(*
Copyrights	: Precision Systems Engineering
Author		: ADBO
Date		: 07/2022
Description	: This function block extends standard functionality of FB_FixtureCore with platform pusher and product holder.
*)
FUNCTION_BLOCK FB_Fixture EXTENDS FB_FixtureJig
VAR CONSTANT
	(* Fixture platform cylinder default setup *)
	sCOVER_PUSHER_NAME						: STRING	:= 'Cover Pusher';	(* Platform pusher name *)
	tCOVER_PUSHER_OPEN_TIMEOUT				: TIME 		:= T#5S;			(* Platform pusher opening timeout *)
	tCOVER_PUSHER_CLOSE_TIMEOUT				: TIME 		:= T#5S;			(* Platform pusher closing timeout *)
	tCOVER_PUSHER_MOVE_DELAY 				: TIME 		:= T#0MS;			(* Platform pusher delay after position change *)
	
	(* Fixture product holder default setup *)
	sCLAMP_NAME								: STRING 	:= 'Clamp Pusher';	(* Product holder name *)
	tCLAMP_OPEN_TIMEOUT						: TIME 		:= T#5S;			(* Product holder opening timeout *)
	tCLAMP_CLOSE_TIMEOUT					: TIME 		:= T#5S;			(* Product holder closing timeout *)
	tCLAMP_MOVE_DELAY 						: TIME 		:= T#300MS;//750MS	(* Product holder delay after position change *)
	
	(* Norm loading keywords *)
	sNORM_LOAD_COMMAND						: STRING := 'LDNORM:';			(* Load norm command send from PLC to UTU*)
	sNORM_GSAMPLE_MEASURE_COMMAND			: STRING := 'MeasGSample';		(* Measure Golden sample command send from PLC to UTU after loading new norm *)	
	sNORM_LOAD_SUCCESS 						: STRING := 'OK';				(* Response from UTU: norm loaded successfull *)
	sNORM_LOAD_FAIL							: STRING := 'Fail';				(* Response from UTU: norm load failed *)
	sNORM_GS_REQUEST						: STRING := 'GS:';				(* UTU requests golden sample *)
 	
	(* UTU STATUS *)
	sUTU_STATUS_OK							: STRING := 'OK';
	sUTU_STATUS_NOK							: STRING := 'NOK';
	sUTU_STATUS_bBusy						: STRING := 'bBusy';
	sUTU_STATUS_BCHECKSETUP					: STRING := 'bCheckSetup';
	
	(* Measurement keywords *)
	sMEASUREMENT_START_COMMAND				: STRING := 'bStart$R$N';		(* Start measurement command send from PLC to UTU*)
	
	sMEASUREMENT_BUSY						: STRING := 'bBusy';			(* Response from UTU: measurement started *)
	sMEASUREMENT_FINISHED					: STRING := (*'bReady'; //*)'bDone';			(* Response from UTU: measurement passed *)
	sMEASUREMENT_GOOD_PRODUCT				: STRING := 'bGood';			(* Response from UTU: good product *)
	sMEASUREMENT_REWORK						: STRING := 'bRework';			(* Perform remeasurement of same product *)
	sMEASUREMENT_REMEASURE					: STRING := 'bRemeasure';		(* Perform remeasurement of same product *)
	sMEASUREMENT_ERROR_THD					: STRING := 'bTHDReject';		(* Response from UTU: measurement failed with THD error*)
	sMEASUREMENT_ERROR_PHASE				: STRING := 'bPhaseReject';		(* Response from UTU: measurement failed with PHASE error*)
	sMEASUREMENT_ERROR_SSPL					: STRING := 'bSSPLReject';		(* Response from UTU: measurement failed with SSPL error*)
	sMEASUREMENT_ERROR_RUBBING				: STRING := 'bRubReject';		(* Response from UTU: measurement failed with RUBBING error*)
	sMEASUREMENT_ERROR_IMP					: STRING := 'bImpReject';		(* Response from UTU: measurement failed with INP error*)
	sMEASUREMENT_ERROR_HFA					: STRING := 'bHFAReject';		(* Response from UTU: measurement failed with HFA error*)
	sMEASUREMENT_ERROR_SPL					: STRING := 'bSPLReject';		(* Response from UTU: measurement failed with SPL error*)
	sMEASUREMENT_ERROR_CONNECTION			: STRING := 'bRejectConnect';	(* Response from UTU: measurement failed with connection problems *)
	sMEASUREMENT_ERROR_OTHER				: STRING := 'bReject';			(* Response from UTU: measurement failed *)
	sMEASUREMENT_FINISH_BATCH				: STRING := 'bFinishBatch';		(* Response from UTU: Batch END *)
	sMEASUREMENT_READY						: STRING := 'bReady';
END_VAR
VAR
	(* Auxilary command bits *)
	bCoverActive 							: BOOL;
	bCoverHome 								: BOOL;
	bClampHold 								: BOOL;
	bClampRelease 							: BOOL;
	bCoverActiveAndJigOpen					: BOOL;
	bCoverHomeAndJigClose					: BOOL;
	bLoadNorm								: BOOL;
//	bGSampleMeasure							: BOOL;
//	bGoldenSampelReadyToMeasure				: BOOL;		(* Robot gived Golden sample to Fixture *)
	
	(* Parameters *)
	sProductType							: STRING;
	sProductQuantity						: STRING;
	
	//new
	sConfig									: STRING;
	iAmount									: UINT;
	sPO										: STRING;
	sBatch									: STRING;
	sOPID									: STRING;
	
	(* Status flags *)
	bNormLoaded								: BOOL;
	bBatchEnd								: BOOL;
	bGSampleMeasureRequested				: BOOL;
	bReMeasure								: BOOL;
	bGSampleMeasurmentDone					: BOOL;
	eNormLoadResult							: E_FixtureLoadNormResult;
	eMeasurementResultExt					: E_FixtureMeasurementResultExt;
	
	(* State machines *)
	eFcqFixtureStateInit					: E_FixtureStateInit;
	eFcqFixtureStateAbort					: E_FixtureStateAbort;
	eFcqFixtrueStateReset					: E_FixtureStateReset;
	eFcqFixtureState						: E_FixtureState;
	eFcqFixtureStateLoadNorm				: E_FixtureStateLoadNorm;
	eFcqFixtureStateGSampleMeas				: E_FcqFixtureStateGSampleMeas;
	eFcqFixtureStateMeasurement 			: E_FixtureStateMeasurement;
	eFcqFixtureStateMeasurementDataExchange	: E_FixtureStateMeasurementDataExchange;
	
	eGoldenSampleResult 					: E_GoldenSampleState;
	
	iGsampleId : USINT;
	
	
	(* FB's *)
	fbCover									: FB_DoubleCoilCylinder;		(*  *)
	fbClamp									: FB_FixtureClamp;				(*  *)
	
END_VAR

IF bFirstCycle THEN
	fbCover.MR_FirstCycle(	sName 					:= CONCAT(STR1 :=THIS^.sName, STR2:= sCOVER_PUSHER_NAME),
							sHomeSensorModuleType	:= '?',
							sHomeSensorPortID		:= '?',
							sActiveSensorModuleType	:= '?',
							sActiveSensorPortID		:= '?',
							tGoHomeTimeout 			:= tCOVER_PUSHER_OPEN_TIMEOUT,
							tGoActiveTimeout 		:= tCOVER_PUSHER_CLOSE_TIMEOUT,
							tDelay					:= tCOVER_PUSHER_MOVE_DELAY);
									
	fbClamp.MR_FirstCycle(	sName 					:= CONCAT(STR1 := THIS^.sName, STR2:= sCLAMP_NAME),
							sHomeSensorModuleType	:= '?',
							sHomeSensorPortID		:= '?',
							sActiveSensorModuleType := '?',
							sActiveSensorPortID		:= '?',
							tGoHomeTimeout 			:= tCLAMP_OPEN_TIMEOUT,
							tGoActiveTimeout 		:= tCLAMP_CLOSE_TIMEOUT,
							tDelay					:= tCLAMP_MOVE_DELAY);							
END_IF

(* Run parent main implementation *)
SUPER^();

(* Update status flags*)
bError := bError OR fbClamp.Error OR fbCover.Error;
//IF bError THEN
//	bBusy := FALSE;
//END_IF

(* Run product holder cylinder instance *)
fbClamp();

(* Run fixture platform cylinder instance *)
fbCover();

PROPERTY BatchEnd : REFERENCE TO BOOL
GET
BatchEnd REF= bBatchEnd;
END_GET
END_PROPERTY

PROPERTY ClampHold : REFERENCE TO BOOL
GET
ClampHold REF= fbClamp.PositionActive;
//ClampHold := NOT fbClamp.PositionActive;
END_GET
END_PROPERTY

PROPERTY ClampSimulation : BOOL
GET
ClampSimulation := fbClamp.Simulation;
END_GET
SET
fbClamp.Simulation := ClampSimulation;
END_SET
END_PROPERTY

PROPERTY CoverPositionActive : REFERENCE TO BOOL
GET
CoverPositionActive REF= fbCover.PositionActive;
END_GET
END_PROPERTY

PROPERTY CoverPositionHome : REFERENCE TO BOOL
GET
CoverPositionHome REF= fbCover.PositionHome;
END_GET
END_PROPERTY

PROPERTY CoverSimulation : BOOL
GET
CoverSimulation := fbCover.Simulation;
END_GET
SET
fbCover.Simulation := CoverSimulation;
END_SET
END_PROPERTY

PROPERTY GoldenSampleMeasDone : REFERENCE TO BOOL
GET
GoldenSampleMeasDone REF= bGSampleMeasurmentDone;
END_GET
END_PROPERTY

PROPERTY GoldenSampleMeasRequested : REFERENCE TO BOOL
GET
GoldenSampleMeasRequested REF= bGSampleMeasureRequested;
END_GET
END_PROPERTY

PROPERTY GoldenSampleResult : REFERENCE TO E_GoldenSampleState
GET
GoldenSampleResult REF= eGoldenSampleResult;
END_GET
END_PROPERTY

PROPERTY GSampleId : REFERENCE TO USINT
GET
GSampleId REF= iGsampleId;
END_GET
END_PROPERTY

METHOD PROTECTED M_MeasurementClient : BOOL
VAR_INST
	tonMeasSimulation : TON;
END_VAR
CASE eFixtureStateMeasure OF
	UNIVERSAL_FIXTURE_MEASURE_SEND_DATA:
		sSendData := sMEASUREMENT_START_COMMAND;
		FUN_StringToTcpBufferData(sMessageAddr := ADR(sSendData), stSendDataAddr := ADR(stSendData));
		fbTcpClient.MR_AppendToSendBuffer(stData := stSendData);
		
		eFixtureStateMeasure := UNIVERSAL_FIXTURE_MEASURE_RECIVE_DATA;
		eFcqFixtureStateMeasurementDataExchange := FIXTURE_MEASURE_DATA_EXCHANGING_WAIT_FOR_BUSY;
		
	UNIVERSAL_FIXTURE_MEASURE_RECIVE_DATA:
		stReciveData := fbTcpClient.NextRecivedMessage;
		
		IF stReciveData.iLength > 0 THEN
			FUN_TcpBufferDataToString(sMessageAddr := ADR(sRecivedData), stReturnDataAddr := ADR(stReciveData));
		END_IF
		
			CASE eFcqFixtureStateMeasurementDataExchange OF
				FIXTURE_MEASURE_DATA_EXCHANGING_WAIT_FOR_BUSY:
					IF MEMCMP(ADR(sRecivedData),ADR(sMEASUREMENT_BUSY),INT_TO_UDINT(LEN(sMEASUREMENT_BUSY))) = 0 THEN
						fbTcpClient.MR_ClearReciveBuffer();
						eFcqFixtureStateMeasurementDataExchange := FIXTURE_MEASURE_DATA_EXCHANGING_WAIT_FOR_FISNISH;
					//	eFcqFixtureStateMeasurementDataExchange := FIXTURE_MEASURE_DATA_EXCHANGING_PROCCESS_RESULTS;
					END_IF
				
				FIXTURE_MEASURE_DATA_EXCHANGING_WAIT_FOR_FISNISH:
					IF (MEMCMP(ADR(sRecivedData),ADR(sMEASUREMENT_FINISHED),INT_TO_UDINT(LEN(sMEASUREMENT_FINISHED))) = 0) OR (FIND(sRecivedData,sMEASUREMENT_FINISHED) > 0) THEN
						IF bReMeasure THEN
							fbTcpClient.MR_ClearReciveBuffer();
							eFixtureStateMeasure := UNIVERSAL_FIXTURE_MEASURE_SEND_DATA;
							eFcqFixtureStateMeasurementDataExchange := FIXTURE_MEASURE_DATA_EXCHANGING_WAIT_FOR_BUSY;
						ELSE
							eFcqFixtureStateMeasurementDataExchange := FIXTURE_MEASURE_DATA_EXCHANGING_PROCCESS_RESULTS;
//							eFcqFixtureStateMeasurementDataExchange := FIXTURE_MEASURE_DATA_EXCHANGING_DONE;//
						END_IF	
					END_IF
				
				FIXTURE_MEASURE_DATA_EXCHANGING_PROCCESS_RESULTS:
					(* Good product *)
					IF (MEMCMP(ADR(sRecivedData),ADR(sMEASUREMENT_GOOD_PRODUCT),INT_TO_UDINT(LEN(sMEASUREMENT_GOOD_PRODUCT))) = 0) OR (FIND(sRecivedData,sMEASUREMENT_GOOD_PRODUCT) > 0) THEN
						IF bUseLogger THEN
							sLoggerMessage := CONCAT(sLoggerMessage,sMEASUREMENT_GOOD_PRODUCT);
							fbMeasurementLogger.MR_AddLogs(sLoggerMessage);
						END_IF
						fbTcpClient.MR_ClearReciveBuffer();
						eSampleResult := UNIVERSAL_FIXTURE_SAMPLE_ACCEPTED;
						eMeasurementResultExt := FIXTURE_MEASUREMENT_RESULT_GOOD;
						eFcqFixtureStateMeasurementDataExchange := FIXTURE_MEASURE_DATA_EXCHANGING_DONE;
//						eFcqFixtureStateMeasurementDataExchange := FIXTURE_MEASURE_DATA_EXCHANGING_WAIT_FOR_FISNISH; //

					(* Bad product - rework *)
					ELSIF (MEMCMP(ADR(sRecivedData),ADR(sMEASUREMENT_REWORK),INT_TO_UDINT(LEN(sMEASUREMENT_REWORK))) = 0) OR (FIND(sRecivedData,sMEASUREMENT_REWORK) > 0) THEN
						IF bUseLogger THEN
							sLoggerMessage := CONCAT(sLoggerMessage,sMEASUREMENT_REWORK);
							fbMeasurementLogger.MR_AddLogs(sLoggerMessage);
						END_IF
						fbTcpClient.MR_ClearReciveBuffer();
						eSampleResult := UNIVERSAL_FIXTURE_SAMPLE_REJECTED;
						eMeasurementResultExt := FIXTURE_MEASUREMENT_RESULT_REWORK;
						eFcqFixtureStateMeasurementDataExchange := FIXTURE_MEASURE_DATA_EXCHANGING_DONE;
//						eFcqFixtureStateMeasurementDataExchange := FIXTURE_MEASURE_DATA_EXCHANGING_WAIT_FOR_FISNISH; //
						
						
					(* Bad product - remeaseure *)
					ELSIF (MEMCMP(ADR(sRecivedData),ADR(sMEASUREMENT_REMEASURE),INT_TO_UDINT(LEN(sMEASUREMENT_REMEASURE))) = 0) OR (FIND(sRecivedData,sMEASUREMENT_REMEASURE) > 0) THEN
						fbTcpClient.MR_ClearSendBuffer();
						fbTcpClient.MR_ClearReciveBuffer();
//						bReMeasure := TRUE;
//						eFcqFixtureStateMeasurementDataExchange :=FIXTURE_MEASURE_DATA_EXCHANGING_WAIT_FOR_FISNISH;
						eFixtureStateMeasure := UNIVERSAL_FIXTURE_MEASURE_SEND_DATA;
						eFcqFixtureStateMeasurementDataExchange := FIXTURE_MEASURE_DATA_EXCHANGING_WAIT_FOR_BUSY;
						
					(* Bad product - connection *)	
					ELSIF (MEMCMP(ADR(sRecivedData),ADR(sMEASUREMENT_ERROR_CONNECTION),INT_TO_UDINT(LEN(sMEASUREMENT_ERROR_CONNECTION))) = 0) OR  (FIND(sRecivedData,sMEASUREMENT_ERROR_CONNECTION) > 0)  THEN
						IF bUseLogger THEN
							sLoggerMessage := CONCAT(sLoggerMessage,sMEASUREMENT_ERROR_CONNECTION);
							fbMeasurementLogger.MR_AddLogs(sLoggerMessage);
						END_IF
						fbTcpClient.MR_ClearReciveBuffer();
						eSampleResult := UNIVERSAL_FIXTURE_SAMPLE_REJECTED;
						eMeasurementResultExt := FIXTURE_MEASUREMENT_RESULT_CONNECT;
						eFcqFixtureStateMeasurementDataExchange := FIXTURE_MEASURE_DATA_EXCHANGING_DONE;
//						eFcqFixtureStateMeasurementDataExchange := FIXTURE_MEASURE_DATA_EXCHANGING_WAIT_FOR_FISNISH; //
					
					(* Bad product - THD *)
					ELSIF (MEMCMP(ADR(sRecivedData),ADR(sMEASUREMENT_ERROR_THD),INT_TO_UDINT(LEN(sMEASUREMENT_ERROR_THD))) = 0) OR (FIND(sRecivedData,sMEASUREMENT_ERROR_THD) > 0)  THEN
						IF bUseLogger THEN
							sLoggerMessage := CONCAT(sLoggerMessage,sMEASUREMENT_ERROR_THD);
							fbMeasurementLogger.MR_AddLogs(sLoggerMessage);
						END_IF
						fbTcpClient.MR_ClearReciveBuffer();
						eSampleResult := UNIVERSAL_FIXTURE_SAMPLE_REJECTED;
						eMeasurementResultExt := (*FIXTURE_MEASUREMENT_RESULT_REWORK;*)FIXTURE_MEASUREMENT_RESULT_THD;
						eFcqFixtureStateMeasurementDataExchange := FIXTURE_MEASURE_DATA_EXCHANGING_DONE;
//						eFcqFixtureStateMeasurementDataExchange := FIXTURE_MEASURE_DATA_EXCHANGING_WAIT_FOR_FISNISH; //
					
					(* Bad product - PHASE *)
					ELSIF (MEMCMP(ADR(sRecivedData),ADR(sMEASUREMENT_ERROR_PHASE),INT_TO_UDINT(LEN(sMEASUREMENT_ERROR_PHASE))) = 0) OR (FIND(sRecivedData,sMEASUREMENT_ERROR_PHASE) > 0) THEN
						IF bUseLogger THEN
							sLoggerMessage := CONCAT(sLoggerMessage,sMEASUREMENT_ERROR_PHASE);
							fbMeasurementLogger.MR_AddLogs(sLoggerMessage);
						END_IF
						fbTcpClient.MR_ClearReciveBuffer();
						eSampleResult := UNIVERSAL_FIXTURE_SAMPLE_REJECTED;
						eMeasurementResultExt := FIXTURE_MEASUREMENT_RESULT_PHASE;
						eFcqFixtureStateMeasurementDataExchange := FIXTURE_MEASURE_DATA_EXCHANGING_DONE;
//						eFcqFixtureStateMeasurementDataExchange := FIXTURE_MEASURE_DATA_EXCHANGING_WAIT_FOR_FISNISH; //
					
					(* Bad product - SSPL *)
					ELSIF (MEMCMP(ADR(sRecivedData),ADR(sMEASUREMENT_ERROR_SSPL),INT_TO_UDINT(LEN(sMEASUREMENT_ERROR_SSPL))) = 0) OR (FIND(sRecivedData,sMEASUREMENT_ERROR_SSPL) > 0) THEN
						IF bUseLogger THEN
							sLoggerMessage := CONCAT(sLoggerMessage,sMEASUREMENT_ERROR_SSPL);
							fbMeasurementLogger.MR_AddLogs(sLoggerMessage);
						END_IF
						fbTcpClient.MR_ClearReciveBuffer();
						eSampleResult := UNIVERSAL_FIXTURE_SAMPLE_REJECTED;
						eMeasurementResultExt := FIXTURE_MEASUREMENT_RESULT_SSPL;
						eFcqFixtureStateMeasurementDataExchange := FIXTURE_MEASURE_DATA_EXCHANGING_DONE;
//						eFcqFixtureStateMeasurementDataExchange := FIXTURE_MEASURE_DATA_EXCHANGING_WAIT_FOR_FISNISH; //
					
					(* Bad product - Rubbing *)
					ELSIF (MEMCMP(ADR(sRecivedData),ADR(sMEASUREMENT_ERROR_RUBBING),INT_TO_UDINT(LEN(sMEASUREMENT_ERROR_RUBBING))) = 0) OR (FIND(sRecivedData,sMEASUREMENT_ERROR_RUBBING) > 0) THEN
						IF bUseLogger THEN
							sLoggerMessage := CONCAT(sLoggerMessage,sMEASUREMENT_ERROR_RUBBING);
							fbMeasurementLogger.MR_AddLogs(sLoggerMessage);
						END_IF
						fbTcpClient.MR_ClearReciveBuffer();
						eSampleResult := UNIVERSAL_FIXTURE_SAMPLE_REJECTED;
						eMeasurementResultExt := FIXTURE_MEASUREMENT_RESULT_RUBBING;
						eFcqFixtureStateMeasurementDataExchange := FIXTURE_MEASURE_DATA_EXCHANGING_DONE;
//						eFcqFixtureStateMeasurementDataExchange := FIXTURE_MEASURE_DATA_EXCHANGING_WAIT_FOR_FISNISH; //
					
					(* Bad product - IMP *)
					ELSIF (MEMCMP(ADR(sRecivedData),ADR(sMEASUREMENT_ERROR_IMP),INT_TO_UDINT(LEN(sMEASUREMENT_ERROR_IMP))) = 0) OR (FIND(sRecivedData,sMEASUREMENT_ERROR_IMP) > 0) THEN
						IF bUseLogger THEN
							sLoggerMessage := CONCAT(sLoggerMessage,sMEASUREMENT_ERROR_IMP);
							fbMeasurementLogger.MR_AddLogs(sLoggerMessage);
						END_IF
						fbTcpClient.MR_ClearReciveBuffer();
						eSampleResult := UNIVERSAL_FIXTURE_SAMPLE_REJECTED;
						eMeasurementResultExt := FIXTURE_MEASUREMENT_RESULT_IMP;
						eFcqFixtureStateMeasurementDataExchange := FIXTURE_MEASURE_DATA_EXCHANGING_DONE;
//						eFcqFixtureStateMeasurementDataExchange := FIXTURE_MEASURE_DATA_EXCHANGING_WAIT_FOR_FISNISH; //
					
					(* Bad product - HFA *)
					ELSIF (MEMCMP(ADR(sRecivedData),ADR(sMEASUREMENT_ERROR_HFA),INT_TO_UDINT(LEN(sMEASUREMENT_ERROR_HFA))) = 0) OR (FIND(sRecivedData,sMEASUREMENT_ERROR_HFA) > 0) THEN
						IF bUseLogger THEN
							sLoggerMessage := CONCAT(sLoggerMessage,sMEASUREMENT_ERROR_HFA);
							fbMeasurementLogger.MR_AddLogs(sLoggerMessage);
						END_IF
						fbTcpClient.MR_ClearReciveBuffer();
						eSampleResult := UNIVERSAL_FIXTURE_SAMPLE_REJECTED;
						eMeasurementResultExt := FIXTURE_MEASUREMENT_RESULT_HFA;
						eFcqFixtureStateMeasurementDataExchange := FIXTURE_MEASURE_DATA_EXCHANGING_DONE;
//						eFcqFixtureStateMeasurementDataExchange := FIXTURE_MEASURE_DATA_EXCHANGING_WAIT_FOR_FISNISH; //
						
					(* Bad product - SPL *)
					ELSIF (MEMCMP(ADR(sRecivedData),ADR(sMEASUREMENT_ERROR_OTHER),INT_TO_UDINT(LEN(sMEASUREMENT_ERROR_OTHER))) = 0) OR (FIND(sRecivedData,sMEASUREMENT_ERROR_OTHER) > 0) THEN
						IF bUseLogger THEN
							sLoggerMessage := CONCAT(sLoggerMessage,sMEASUREMENT_ERROR_SPL);
							fbMeasurementLogger.MR_AddLogs(sLoggerMessage);
						END_IF
						fbTcpClient.MR_ClearReciveBuffer();
						eSampleResult := UNIVERSAL_FIXTURE_SAMPLE_REJECTED;
						eMeasurementResultExt := FIXTURE_MEASUREMENT_RESULT_SPL;
						eFcqFixtureStateMeasurementDataExchange := FIXTURE_MEASURE_DATA_EXCHANGING_DONE;
//						eFcqFixtureStateMeasurementDataExchange := FIXTURE_MEASURE_DATA_EXCHANGING_WAIT_FOR_FISNISH; //
					
					ELSIF (MEMCMP(ADR(sRecivedData),ADR(sMEASUREMENT_ERROR_OTHER),INT_TO_UDINT(LEN(sMEASUREMENT_ERROR_OTHER))) = 0) OR (FIND(sRecivedData,sMEASUREMENT_ERROR_OTHER) > 0)  THEN
						IF bUseLogger THEN
							sLoggerMessage := CONCAT(sLoggerMessage,sMEASUREMENT_ERROR_OTHER);
							fbMeasurementLogger.MR_AddLogs(sLoggerMessage);
						END_IF
						fbTcpClient.MR_ClearReciveBuffer();
						eSampleResult := UNIVERSAL_FIXTURE_SAMPLE_REJECTED;
						eMeasurementResultExt := FIXTURE_MEASUREMENT_RESULT_REJECT_OTHER;
						eFcqFixtureStateMeasurementDataExchange := FIXTURE_MEASURE_DATA_EXCHANGING_DONE;
					
					ELSIF (MEMCMP(ADR(sRecivedData),ADR(sMEASUREMENT_READY),INT_TO_UDINT(LEN(sMEASUREMENT_READY))) = 0) OR (FIND(sRecivedData,sMEASUREMENT_READY) > 0)  THEN 
						eFcqFixtureStateMeasurementDataExchange := FIXTURE_MEASURE_DATA_EXCHANGING_DONE;	
					END_IF
					
				FIXTURE_MEASURE_DATA_EXCHANGING_DONE:
					IF (MEMCMP(ADR(sRecivedData),ADR(sMEASUREMENT_READY),INT_TO_UDINT(LEN(sMEASUREMENT_READY))) = 0) OR (FIND(sRecivedData,sMEASUREMENT_READY) > 0) THEN
						eFixtureStateMeasure := UNIVERSAL_FIXTURE_MEASURE_DONE;
					END_IF
			END_CASE		
	//	END_IF
	
	UNIVERSAL_FIXTURE_MEASURE_DONE:
		IF 	(MEMCMP(ADR(sRecivedData),ADR(sMEASUREMENT_FINISH_BATCH),INT_TO_UDINT(LEN(sMEASUREMENT_FINISH_BATCH))) = 0) OR (FIND(sRecivedData,sMEASUREMENT_FINISH_BATCH) > 0) THEN
			bBatchEnd := TRUE;
		END_IF
		fbTcpClient.MR_ClearAllBuffers();
		eFixtureState := UNIVERSAL_FIXTURE_METHOD_DONE;
		
END_CASE
(*
tonMeasSimulation(IN := TRUE, PT := T#2500MS);
IF tonMeasSimulation.Q THEN
	tonMeasSimulation(IN := FALSE);
	eSampleResult := UNIVERSAL_FIXTURE_SAMPLE_ACCEPTED;
	eMeasurementResultExt := FIXTURE_MEASUREMENT_RESULT_GOOD;
	eFixtureState := UNIVERSAL_FIXTURE_METHOD_DONE;
END_IF
*)
END_METHOD

PROPERTY MeasurementResultExt : REFERENCE TO E_FixtureMeasurementResultExt
GET
MeasurementResultExt REF= eMeasurementResultExt;
END_GET
END_PROPERTY

METHOD MR_ClampHold : BOOL
VAR_INPUT
END_VAR
IF eFixtureState = UNIVERSAL_FIXTURE_IDLE AND NOT fbClamp.PositionActive THEN
	bBusy := TRUE;
	bClampHold := TRUE;
	MR_ClampHold := FALSE;
	eFixtureState := UNIVERSAL_FIXTURE_EXTENSION;
	eFcqFixtureState := FIXTURE_EXTENSION_CLAMP_HOLD;
	fbMachineLogger.MR_AddLogs(CONCAT(sName,' : product hold'));
	
ELSIF eFcqFixtureState = FIXTURE_EXTENSION_CLAMP_HOLD_DONE THEN
	bClampHold := FALSE;
	MR_ClampHold := TRUE;
	fbMachineLogger.MR_AddLogs(CONCAT(sName,' : product hold done'));
	
END_IF
END_METHOD

METHOD MR_ClampRelease : BOOL
VAR_INPUT
END_VAR
IF eFixtureState = UNIVERSAL_FIXTURE_IDLE AND fbClamp.PositionActive THEN
	bBusy := TRUE;
	bClampRelease := TRUE;
	MR_ClampRelease := FALSE;
	eFixtureState := UNIVERSAL_FIXTURE_EXTENSION;
	eFcqFixtureState := FIXTURE_EXTENSION_CLAMP_RELEASE;
	fbMachineLogger.MR_AddLogs(CONCAT(sName,' : product release'));
	
ELSIF eFcqFixtureState = FIXTURE_EXTENSION_CLAMP_RELEASE_DONE THEN
	bClampRelease := FALSE;
	MR_ClampRelease := TRUE;
	fbMachineLogger.MR_AddLogs(CONCAT(sName,' : product release done'));
	
END_IF
END_METHOD

METHOD MR_CoverActive : BOOL
VAR_INPUT
END_VAR
IF eFixtureState = UNIVERSAL_FIXTURE_IDLE AND NOT fbCover.PositionActive THEN
	bBusy := TRUE;
	bCoverActive := TRUE;
	MR_CoverActive := FALSE;
	eFixtureState := UNIVERSAL_FIXTURE_EXTENSION;
	eFcqFixtureState := FIXTURE_EXTENSION_COVER_ACTIVE;
	fbMachineLogger.MR_AddLogs(CONCAT(sName,' : platform go active'));
	
ELSIF eFcqFixtureState = FIXTURE_EXTENSION_COVER_ACTIVE_DONE THEN
	bCoverActive := FALSE;
	MR_CoverActive := TRUE;
	fbMachineLogger.MR_AddLogs(CONCAT(sName,' : platform go active done'));
	
END_IF
END_METHOD

METHOD MR_CoverActiveAndJigOpen : BOOL
VAR_INPUT
END_VAR
//IF eFixtureState = UNIVERSAL_FIXTURE_IDLE AND (NOT fbCover.PositionActive AND NOT THIS^.SocketOpen) THEN
IF eFixtureState = UNIVERSAL_FIXTURE_IDLE AND (NOT fbCover.PositionActive OR NOT THIS^.SocketOpen) THEN
	bBusy := TRUE;
	bCoverActiveAndJigOpen := TRUE;
	MR_CoverActiveAndJigOpen := FALSE;
	eFixtureState := UNIVERSAL_FIXTURE_EXTENSION;
	eFcqFixtureState := FIXTURE_EXTENSION_COVER_ACTIVE_AND_JIG_OPEN;
	fbMachineLogger.MR_AddLogs(CONCAT(sName,' : platform go active and open'));
	
ELSIF eFcqFixtureState = FIXTURE_EXTENSION_COVER_ACTIVE_AND_JIG_OPEN_DONE THEN
	bCoverActiveAndJigOpen := FALSE;
	MR_CoverActiveAndJigOpen := TRUE;
	fbMachineLogger.MR_AddLogs(CONCAT(sName,' : platform go active and open done'));
	
END_IF
END_METHOD

METHOD MR_CoverHome : BOOL
VAR_INPUT
END_VAR
IF eFixtureState = UNIVERSAL_FIXTURE_IDLE AND NOT fbCover.PositionHome THEN
	bBusy := TRUE;
	bCoverHome := TRUE;
	MR_CoverHome := FALSE;
	eFixtureState := UNIVERSAL_FIXTURE_EXTENSION;
	eFcqFixtureState := FIXTURE_EXTENSION_COVER_HOME;
	fbMachineLogger.MR_AddLogs(CONCAT(sName,' : platform go home'));
	
ELSIF eFcqFixtureState = FIXTURE_EXTENSION_COVER_HOME_DONE THEN
	bCoverHome := FALSE;
	MR_CoverHome := TRUE;
	fbMachineLogger.MR_AddLogs(CONCAT(sName,' : platform go home done'));
	
END_IF
END_METHOD

METHOD MR_CoverHomeAndJigClose : BOOL
VAR_INPUT
END_VAR
//IF eFixtureState = UNIVERSAL_FIXTURE_IDLE AND NOT fbCover.PositionHome AND THIS^.SocketOpen THEN
IF eFixtureState = UNIVERSAL_FIXTURE_IDLE AND (NOT fbCover.PositionHome OR THIS^.SocketOpen) THEN
	bBusy := TRUE;
	bCoverHomeAndJigClose := TRUE;
	MR_CoverHomeAndJigClose := FALSE;
	eFixtureState := UNIVERSAL_FIXTURE_EXTENSION;
	eFcqFixtureState := FIXTURE_EXTENSION_COVER_HOME_AND_JIG_CLOSE;
	fbMachineLogger.MR_AddLogs(CONCAT(sName,' : platform go home and close'));
	
ELSIF eFcqFixtureState = FIXTURE_EXTENSION_COVER_HOME_AND_JIG_CLOSE_DONE THEN
	bCoverHomeAndJigClose := FALSE;
	MR_CoverHomeAndJigClose := TRUE;
	fbMachineLogger.MR_AddLogs(CONCAT(sName,' : platform go home and close done'));
	
END_IF
END_METHOD

METHOD MR_GSampleMeas : BOOL
VAR_INPUT
END_VAR
//IF eNormLoadResult = FIXTURE_NORM_LOAD_GOLDEN_SAMPLE_NEEDED AND eFcqFixtureStateLoadNorm = FIXTURE_LOADING_NORM_GOLDEN_SAMPLE_WAIT_FOR_END THEN
IF eNormLoadResult = FIXTURE_NORM_LOAD_GOLDEN_SAMPLE_NEEDED AND eFixtureState = UNIVERSAL_FIXTURE_IDLE THEN
	bBusy := TRUE;
	bGSampleMeasurmentDone := FALSE;	
	MR_GSampleMeas := FALSE;
//	bGSampleMeasure := TRUE;
	eGoldenSampleResult := GS_STATUS_UNKNOWN;
	eFixtureState := UNIVERSAL_FIXTURE_EXTENSION;
	eFcqFixtureState := FIXTURE_EXTENSION_GOLDEN_SAMPLE_MEASURE;
	eFcqFixtureStateGSampleMeas := FIXTURE_GOLDEN_SAMPLE_SEND_MEASURE_COMMAND;
	fbMachineLogger.MR_AddLogs(CONCAT(sName,' : Golden Sample measurment requested'));
	
	
ELSIF eFcqFixtureState = FIXTURE_EXTENSION_GOLDEN_SAMPLE_MEASURE_DONE THEN
	bBusy := FALSE;
	MR_GSampleMeas := TRUE;
	eFixtureState := UNIVERSAL_FIXTURE_EXTENSION;
	eFcqFixtureState := FIXTURE_EXTENSION_LOAD_NORM;
	//eFcqFixtureStateLoadNorm := FIXTURE_LOADING_NORM_WAIT_FOR_RESPONSE;
	//fbMachineLogger.MR_AddLogs(CONCAT(sName,' : Golden Sample  '));
	fbMachineLogger.MR_AddLogs(CONCAT(sName,CONCAT(' : Golden Sample ID: ',CONCAT(UDINT_TO_STRING(iGsampleId),' measurment done'))));
	bGSampleMeasurmentDone := TRUE;
END_IF
END_METHOD

METHOD MR_LoadNorm : BOOL
VAR_INPUT
	sConfig				: STRING;
	iAmount				: UINT;
	sPO					: STRING;
	sBatch				: STRING;
	sOPID				: STRING;
//	sProductType 		: STRING;	(* Name of product possesed from MES*)
//	sProductQuantity	: STRING;	(* Product quantity *)
END_VAR
IF eFixtureState = UNIVERSAL_FIXTURE_IDLE THEN
	THIS^.sConfig := sConfig;
	THIS^.iAmount := iAmount;
	THIS^.sPO := sPO;
	THIS^.sBatch := sBatch;
	THIS^.sOPID := sOPID;
	
(*	OLD
	THIS^.sProductType := sProductType;
	THIS^.sProductQuantity := sProductQuantity;
*)	
	bNormLoaded := FALSE;
	eNormLoadResult := FIXTURE_NORM_LOAD_UNKNOWN;
//	bLoadNorm := TRUE;
	MR_LoadNorm := FALSE;
	eFixtureState := UNIVERSAL_FIXTURE_EXTENSION;
	eFcqFixtureState := FIXTURE_EXTENSION_LOAD_NORM;
	eFcqFixtureStateLoadNorm := FIXTURE_LOADING_NORM_SEND_NORM_DATA;
	fbMachineLogger.MR_AddLogs(CONCAT(sName,' : load norm requested'));
	
ELSIF eFcqFixtureState = FIXTURE_EXTENSION_LOAD_NORM_DONE THEN
	bNormLoaded := (*NOT bGSampleMeasureRequested;//*)TRUE;
	MR_LoadNorm := TRUE;
	fbMachineLogger.MR_AddLogs(CONCAT(sName,' : norm loaded '));
	
END_IF
END_METHOD

METHOD MR_Reset : BOOL
VAR_INPUT
END_VAR
IF eFixtureState = UNIVERSAL_FIXTURE_METHOD_DONE THEN
	eFcqFixtrueStateReset:=FIXTURE_RESET_CLAMP;
END_IF
SUPER^.MR_Reset();
END_METHOD

METHOD PROTECTED MS_Aborting
VAR_INPUT
END_VAR
CASE eFcqFixtureStateAbort OF
	FIXTURE_ABORT_CLAMP:
		fbClamp.MR_Abort();
		IF NOT fbClamp.Active THEN
			eFcqFixtureStateAbort := FIXTURE_ABORT_COVER;
		END_IF
		
	FIXTURE_ABORT_COVER:
		fbCover.MR_Abort();
		IF NOT fbCover.Active THEN
			eJigStateAbort := FIXTURE_JIG_ABORT_JIG_PUSHER;
			eFcqFixtureStateAbort := FIXTURE_ABORT_DONE;
		END_IF
		
	FIXTURE_ABORT_DONE:
		SUPER^.MS_Aborting();
		
END_CASE
END_METHOD

METHOD MS_ClampHold
VAR_INPUT
END_VAR
fbClamp.MR_GoActive();
IF fbClamp.PositionActive AND NOT fbClamp.Busy THEN
	eFcqFixtureState := FIXTURE_EXTENSION_CLAMP_HOLD_DONE;
END_IF
END_METHOD

METHOD MS_ClampHoldDone
VAR_INPUT
END_VAR
IF NOT bClampHold THEN
	bBusy := FALSE;
	eFixtureState := UNIVERSAL_FIXTURE_IDLE;
	eFcqFixtureState := FIXTURE_EXTENSION_IDLE;
END_IF
END_METHOD

METHOD MS_ClampRelease
VAR_INPUT
END_VAR
fbClamp.MR_GoHome();
IF NOT fbClamp.PositionActive AND NOT fbClamp.Busy THEN
	eFcqFixtureState := FIXTURE_EXTENSION_CLAMP_RELEASE_DONE;
END_IF
END_METHOD

METHOD MS_ClampReleaseDone
VAR_INPUT
END_VAR
IF NOT bClampRelease THEN
	bBusy := FALSE;
	eFixtureState := UNIVERSAL_FIXTURE_IDLE;
	eFcqFixtureState := FIXTURE_EXTENSION_IDLE;
END_IF
END_METHOD

METHOD MS_CoverActive
VAR_INPUT
END_VAR
fbCover.MR_GoActive();
IF fbCover.PositionActive AND NOT fbCover.Busy THEN
	eFcqFixtureState := FIXTURE_EXTENSION_COVER_ACTIVE_DONE;
END_IF
END_METHOD

METHOD MS_CoverActiveAndJigOpen : BOOL
VAR_INPUT
END_VAR
fbCover.MR_GoActive();
fbJig.MR_GoActive();
IF fbCover.PositionActive AND NOT fbCover.Busy AND
	fbJig.PositionActive AND NOT fbJig.Busy THEN
	eFcqFixtureState := FIXTURE_EXTENSION_COVER_ACTIVE_AND_JIG_OPEN_DONE;
END_IF
END_METHOD

METHOD MS_CoverActiveAndJigOpenDone : BOOL
VAR_INPUT
END_VAR
IF NOT bCoverActiveAndJigOpen THEN
	bBusy := FALSE;
	eFixtureState := UNIVERSAL_FIXTURE_IDLE;
	eFcqFixtureState := FIXTURE_EXTENSION_IDLE;
END_IF
END_METHOD

METHOD MS_CoverActiveDone
VAR_INPUT
END_VAR
IF NOT bCoverActive THEN
	bBusy := FALSE;
	eFixtureState := UNIVERSAL_FIXTURE_IDLE;
	eFcqFixtureState := FIXTURE_EXTENSION_IDLE;
END_IF
END_METHOD

METHOD MS_CoverHome
VAR_INPUT
END_VAR
fbCover.MR_GoHome();
IF fbCover.PositionHome AND NOT fbCover.Busy THEN
	eFcqFixtureState := FIXTURE_EXTENSION_COVER_HOME_DONE;
END_IF
END_METHOD

METHOD MS_CoverHomeAndJigClose : BOOL
VAR_INPUT
END_VAR
fbCover.MR_GoHome();
fbJig.MR_GoHome();
IF fbCover.PositionHome AND NOT fbCover.Busy AND
	fbJig.PositionHome AND NOT fbJig.Busy THEN
	eFcqFixtureState := FIXTURE_EXTENSION_COVER_HOME_AND_JIG_CLOSE_DONE;
END_IF
END_METHOD

METHOD MS_CoverHomeAndJigCloseDone : BOOL
VAR_INPUT
END_VAR
IF NOT bCoverHomeAndJigClose THEN
	bBusy := FALSE;
	eFixtureState := UNIVERSAL_FIXTURE_IDLE;
	eFcqFixtureState := FIXTURE_EXTENSION_IDLE;
END_IF
END_METHOD

METHOD MS_CoverHomeDone
VAR_INPUT
END_VAR
IF NOT bCoverHome THEN
	bBusy := FALSE;
	eFixtureState := UNIVERSAL_FIXTURE_IDLE;
	eFcqFixtureState := FIXTURE_EXTENSION_IDLE;
END_IF
END_METHOD

METHOD PROTECTED MS_Extension
VAR_INPUT
END_VAR
CASE eFcqFixtureState OF
	E_FixtureState.FIXTURE_EXTENSION_IDLE:
		bBusy := FALSE;
		
	E_FixtureState.FIXTURE_EXTENSION_COVER_ACTIVE:
		MS_CoverActive();
		
	E_FixtureState.FIXTURE_EXTENSION_COVER_ACTIVE_DONE:
		MS_CoverActiveDone();
		
	E_FixtureState.FIXTURE_EXTENSION_COVER_HOME:
		MS_CoverHome();
		
	E_FixtureState.FIXTURE_EXTENSION_COVER_HOME_DONE:
		MS_CoverHomeDone();	
	
	E_FixtureState.FIXTURE_EXTENSION_CLAMP_HOLD:
		MS_ClampHold();
		
	E_FixtureState.FIXTURE_EXTENSION_CLAMP_HOLD_DONE:
		MS_ClampHoldDone();
		
	E_FixtureState.FIXTURE_EXTENSION_CLAMP_RELEASE:
		MS_ClampRelease();
		
	E_FixtureState.FIXTURE_EXTENSION_CLAMP_RELEASE_DONE:
		MS_ClampReleaseDone();
	
	FIXTURE_EXTENSION_COVER_ACTIVE_AND_JIG_OPEN:
		MS_CoverActiveAndJigOpen();
		
	FIXTURE_EXTENSION_COVER_ACTIVE_AND_JIG_OPEN_DONE:
		MS_CoverActiveAndJigOpenDone();
		
	FIXTURE_EXTENSION_COVER_HOME_AND_JIG_CLOSE:
		MS_CoverHomeAndJigClose();
		
	FIXTURE_EXTENSION_COVER_HOME_AND_JIG_CLOSE_DONE:
		MS_CoverHomeAndJigCloseDone();
		
	FIXTURE_EXTENSION_LOAD_NORM:
		MS_LoadNorm();
		
	FIXTURE_EXTENSION_LOAD_NORM_DONE:
		MS_LoadNormDone();
		
	FIXTURE_EXTENSION_GOLDEN_SAMPLE_MEASURE:	
		MS_GSampleMeas();
		
	FIXTURE_EXTENSION_GOLDEN_SAMPLE_MEASURE_DONE:
		MS_GSampleMeasDone();
	
END_CASE
END_METHOD

METHOD MS_GSampleMeas : BOOL
bBusy := MEMCMP(ADR(sRecivedData),ADR(sUTU_STATUS_bBusy),INT_TO_UDINT(LEN(sUTU_STATUS_bBusy))) = 0; (*	UTU busy flags *)	
CASE eFcqFixtureStateGSampleMeas OF
	//FIXTURE_GOLDEN_SAMPLE_CLOSE:
	//	fbJig.MR_GoActive();
	//	IF fbJig.PositionActive AND NOT fbJig.Busy THEN
	//		eFcqFixtureStateGSampleMeas := FIXTURE_GOLDEN_SAMPLE_SEND_MEASURE_COMMAND;
	//	END_IF
	
	FIXTURE_GOLDEN_SAMPLE_SEND_MEASURE_COMMAND:
		sSendData := sNORM_GSAMPLE_MEASURE_COMMAND;
		sSendData := CONCAT(sSendData, '$R$N');
		FUN_StringToTcpBufferData(sMessageAddr := ADR(sSendData), stSendDataAddr := ADR(stSendData));
		fbTcpClient.MR_AppendToSendBuffer(stData := stSendData);
		eFcqFixtureStateGSampleMeas := FIXTURE_GOLDEN_SAMPLE_WAIT_FOR_RESPONSE;
		
	FIXTURE_GOLDEN_SAMPLE_WAIT_FOR_RESPONSE:
		stReciveData := fbTcpClient.NextRecivedMessage;
		IF stReciveData.iLength > 0 THEN
			FUN_TcpBufferDataToString(sMessageAddr := ADR(sRecivedData), stReturnDataAddr := ADR(stReciveData));
			(* UTU returns bCheckSetup *)
			IF (MEMCMP(ADR(sRecivedData),ADR(sUTU_STATUS_BCHECKSETUP),INT_TO_UDINT(LEN(sUTU_STATUS_BCHECKSETUP))) = 0) THEN
				IF bUseLogger THEN
					sLoggerMessage := CONCAT(sLoggerMessage,sUTU_STATUS_BCHECKSETUP);
					fbMeasurementLogger.MR_AddLogs(sLoggerMessage);
				END_IF
				eGoldenSampleResult := GS_STATUS_BCHECKSETUP;
				//eNormLoadResult := FIXTURE_NORM_LOAD_FAIL;
				eFcqFixtureStateGSampleMeas := FIXTURE_GOLDEN_SAMPLE_MEASUREMENT_DONE; 
			(* UTU returns NOK *)	
			ELSIF (MEMCMP(ADR(sRecivedData),ADR(sUTU_STATUS_NOK),INT_TO_UDINT(LEN(sUTU_STATUS_NOK))) = 0) THEN
				eFcqFixtureStateGSampleMeas := FIXTURE_GOLDEN_SAMPLE_WAIT_FOR_UTU;
				eGoldenSampleResult := GS_STATUS_NOK;
			(* UTU returns OK *)		
			ELSIF (MEMCMP(ADR(sRecivedData),ADR(sUTU_STATUS_OK),INT_TO_UDINT(LEN(sUTU_STATUS_OK))) = 0) THEN
				IF bUseLogger THEN
					sLoggerMessage := CONCAT(sLoggerMessage,sSAMPLE_ACCEPTED);
					fbMeasurementLogger.MR_AddLogs(sLoggerMessage);
				END_IF
				eGoldenSampleResult := GS_STATUS_OK;
				eFcqFixtureStateGSampleMeas := FIXTURE_GOLDEN_SAMPLE_MEASUREMENT_DONE;		
			END_IF
		END_IF
		
(*	FIXTURE_GOLDEN_SAMPLE_OPEN:
		fbJig.MR_GoHome();
		IF (fbJig.PositionHome AND NOT fbJig.Busy) AND NOT fbCover.PositionHome THEN
 			fbClamp.MR_GoHome(); 			
		ELSE
			fbClamp.MR_GoActive();
		END_IF
		IF fbJig.PositionHome AND fbClamp.PositionHome THEN
			fbCover.MR_GoHome();
		END_IF
				
		IF fbClamp.PositionActive AND NOT fbClamp.Busy AND fbCover.PositionHome AND NOT fbCover.Busy AND 
			fbJig.PositionHome AND NOT fbJig.Busy THEN
			eFcqFixtureStateGSampleMeas := FIXTURE_GOLDEN_SAMPLE_MEASUREMENT_DONE;
		ELSE eFcqFixtureStateGSampleMeas := FIXTURE_GOLDEN_SAMPLE_OPEN;
		END_IF
*)
	FIXTURE_GOLDEN_SAMPLE_WAIT_FOR_UTU:
		stReciveData := fbTcpClient.NextRecivedMessage;
		IF stReciveData.iLength > 0 THEN
			FUN_TcpBufferDataToString(sMessageAddr := ADR(sRecivedData), stReturnDataAddr := ADR(stReciveData));
			IF (MEMCMP(ADR(sRecivedData),ADR(sUTU_STATUS_BCHECKSETUP),INT_TO_UDINT(LEN(sUTU_STATUS_BCHECKSETUP))) = 0) THEN
				IF bUseLogger THEN
					sLoggerMessage := CONCAT(sLoggerMessage,sUTU_STATUS_BCHECKSETUP);
					fbMeasurementLogger.MR_AddLogs(sLoggerMessage);
				END_IF
				eGoldenSampleResult := GS_STATUS_BCHECKSETUP;
				//eNormLoadResult := FIXTURE_NORM_LOAD_FAIL;
				eFcqFixtureStateGSampleMeas := FIXTURE_GOLDEN_SAMPLE_MEASUREMENT_DONE; 
			(* UTU returns bCheckSetup *)
			ELSIF (MEMCMP(ADR(sRecivedData),ADR(sNORM_GS_REQUEST),INT_TO_UDINT(LEN(sNORM_GS_REQUEST))) = 0) OR (FIND(sRecivedData,sNORM_GS_REQUEST) > 0) THEN
				bGSampleMeasureRequested := TRUE;
				iGsampleId := STRING_TO_USINT(LEFT(RIGHT(sRecivedData,2),1));
				IF bUseLogger THEN
					sLoggerMessage := CONCAT(sLoggerMessage,'Golden Sample Test');
					fbMeasurementLogger.MR_AddLogs(sLoggerMessage);
				END_IF
				eFcqFixtureStateGSampleMeas := FIXTURE_GOLDEN_SAMPLE_MEASUREMENT_DONE;
			END_IF
		END_IF	
		
	FIXTURE_GOLDEN_SAMPLE_MEASUREMENT_DONE:
		eFcqFixtureState := FIXTURE_EXTENSION_GOLDEN_SAMPLE_MEASURE_DONE;
		
END_CASE
END_METHOD

METHOD MS_GSampleMeasDone : BOOL
VAR_INPUT
END_VAR
bBusy := FALSE;
//eFixtureState := UNIVERSAL_FIXTURE_EXTENSION;
//eFcqFixtureState := FIXTURE_EXTENSION_LOAD_NORM;
//eFcqFixtureStateLoadNorm := FIXTURE_LOADING_NORM_WAIT_FOR_RESPONSE;
eFixtureState := UNIVERSAL_FIXTURE_IDLE;
eFcqFixtureState := FIXTURE_EXTENSION_IDLE;
bGSampleMeasurmentDone := TRUE;
END_METHOD

METHOD PROTECTED MS_Initializing
VAR_INPUT
END_VAR
CASE eFcqFixtureStateInit OF
	FIXTURE_INIT_CLAMP:
		fbClamp.MR_Init();
		
		IF fbClamp.Active THEN
			eFcqFixtureStateInit := FIXTURE_INIT_COVER;
		END_IF
		
	FIXTURE_INIT_COVER:
		fbCover.MR_Init();
		
		IF fbCover.Active THEN
			eJigStateInit := FIXTURE_JIG_INIT_JIG_PUSHER;
			eFcqFixtureStateInit := FIXTURE_INIT_DONE;
		END_IF
		
	FIXTURE_INIT_DONE:
		SUPER^.MS_Initializing();
		
END_CASE
END_METHOD

METHOD MS_LoadNorm
VAR_INST
	TestTON :	TON;
END_VAR
bBusy := MEMCMP(ADR(sRecivedData),ADR(sUTU_STATUS_bBusy),INT_TO_UDINT(LEN(sUTU_STATUS_bBusy))) = 0; (*	UTU busy flags *)	

		
CASE eFcqFixtureStateLoadNorm OF
	FIXTURE_LOADING_NORM_SEND_NORM_DATA:
		(* Prepare and send data to client *)
		sSendData := CONCAT(STR1 := sNORM_LOAD_COMMAND, 
			STR2 :=	CONCAT(STR1 := sConfig,STR2 := CONCAT(STR1 := ':', 
			STR2 := CONCAT(STR1 := UINT_TO_STRING(iAmount),	STR2 := CONCAT(STR1 := ':',
			STR2 := CONCAT(STR1:= sPO, STR2:= CONCAT(STR1:= ':', 
			STR2 := CONCAT(STR1 := sBatch, STR2 := CONCAT(STR1:= ':',
			STR2 := CONCAT(STR1:=sOPID, STR2:= ':'))))))))));
		
		sSendData := CONCAT(sSendData, '$R$N');
		FUN_StringToTcpBufferData(sMessageAddr := ADR(sSendData), stSendDataAddr := ADR(stSendData));
		fbTcpClient.MR_AppendToSendBuffer(stData := stSendData);
		
		(* Prepare data for logger *)
		IF bUseLogger THEN
			MEMSET(ADR(sLoggerMessage),0,INT_TO_UDINT(LEN(sLoggerMessage)));
			sLoggerMessage := CONCAT(STR1 := 'Load norm request:',STR2 := CONCAT(STR1 := sProductType,STR2 := (*USINT_TO_STRING*)(sProductQuantity)));
		END_IF
		
		eFcqFixtureStateLoadNorm := FIXTURE_LOADING_NORM_WAIT_FOR_RESPONSE;
		
	FIXTURE_LOADING_NORM_WAIT_FOR_RESPONSE:
		stReciveData := fbTcpClient.NextRecivedMessage;
		IF stReciveData.iLength > 0  THEN
		FUN_TcpBufferDataToString(sMessageAddr := ADR(sRecivedData), stReturnDataAddr := ADR(stReciveData));
		(* Norm loading Gold Sample *)
			IF (MEMCMP(ADR(sRecivedData),ADR(sNORM_GS_REQUEST),INT_TO_UDINT(LEN(sNORM_GS_REQUEST))) = 0) OR (FIND(sRecivedData,sNORM_GS_REQUEST) > 0) THEN
				iSampleID := STRING_TO_USINT(LEFT(RIGHT(sRecivedData,2),1));
				bGSampleMeasureRequested := TRUE;
				IF bUseLogger THEN
					sLoggerMessage := CONCAT(sLoggerMessage,'Golden Sample Test');
					fbMeasurementLogger.MR_AddLogs(sLoggerMessage);
				END_IF
				
				bGSampleMeasurmentDone := FALSE;
				bBusy := FALSE;
				eNormLoadResult := FIXTURE_NORM_LOAD_GOLDEN_SAMPLE_NEEDED;
				eFcqFixtureStateLoadNorm := FIXTURE_LOADING_NORM_DONE;
				
//			eFcqFixtureStateLoadNorm :=FIXTURE_LOADING_NORM_GOLDEN_SAMPLE_TEST;
							
//			ELSIF MEMCMP(ADR(sRecivedData),ADR(sUTU_STATUS_NOK),INT_TO_UDINT(LEN(sUTU_STATUS_NOK))) = 0 THEN
//				IF bUseLogger THEN
//					sLoggerMessage := CONCAT(sLoggerMessage,CONCAT('golden sample ID:',CONCAT(USINT_TO_STRING(iGsampleId),'	NOK')));
//					fbMeasurementLogger.MR_AddLogs(sLoggerMessage);
//				END_IF
				
			(* Norm loading successfull *)
			ELSIF MEMCMP(ADR(sRecivedData),ADR(sNORM_LOAD_SUCCESS),INT_TO_UDINT(LEN(sNORM_LOAD_SUCCESS))) = 0 THEN
				IF bUseLogger THEN
					sLoggerMessage := CONCAT(sLoggerMessage,sSAMPLE_ACCEPTED);
					fbMeasurementLogger.MR_AddLogs(sLoggerMessage);
				END_IF
				bGSampleMeasureRequested := FALSE;
				bBusy := FALSE;
				eNormLoadResult := FIXTURE_NORM_LOAD_SUCCESS;
				eFcqFixtureStateLoadNorm := FIXTURE_LOADING_NORM_DONE;
				
				
			(* Norm loading failed *)
			ELSIF (MEMCMP(ADR(sRecivedData),ADR(sNORM_LOAD_FAIL),INT_TO_UDINT(LEN(sNORM_LOAD_FAIL))) = 0) THEN
				IF bUseLogger THEN
					sLoggerMessage := CONCAT(sLoggerMessage,sSAMPLE_REJECTED);
					fbMeasurementLogger.MR_AddLogs(sLoggerMessage);
				END_IF
				bGSampleMeasureRequested := FALSE;
				bBusy := FALSE;
				eNormLoadResult := FIXTURE_NORM_LOAD_FAIL;
				eFcqFixtureStateLoadNorm := FIXTURE_LOADING_NORM_DONE;
			
			(* UTU returns bCheckSetup *)
			ELSIF (MEMCMP(ADR(sRecivedData),ADR(sUTU_STATUS_BCHECKSETUP),INT_TO_UDINT(LEN(sUTU_STATUS_BCHECKSETUP))) = 0) THEN
				IF bUseLogger THEN
					sLoggerMessage := CONCAT(sLoggerMessage,sUTU_STATUS_BCHECKSETUP);
					fbMeasurementLogger.MR_AddLogs(sLoggerMessage);
				END_IF
				bGSampleMeasureRequested := FALSE;
				bBusy := FALSE;
				eNormLoadResult := FIXTURE_NORM_LOAD_FAIL;
				eFcqFixtureStateLoadNorm := FIXTURE_LOADING_NORM_DONE;
			END_IF
		END_IF
			
	FIXTURE_LOADING_NORM_DONE:
		fbTcpClient.MR_ClearAllBuffers();
		eFcqFixtureState := FIXTURE_EXTENSION_LOAD_NORM_DONE;
		
END_CASE
END_METHOD

METHOD MS_LoadNormDone
VAR_INPUT
END_VAR
IF NOT bLoadNorm THEN
	bBusy := FALSE;
	bBatchEnd := FALSE;
	eFixtureState := UNIVERSAL_FIXTURE_IDLE;
	eFcqFixtureState := FIXTURE_EXTENSION_IDLE;
END_IF
END_METHOD

METHOD PROTECTED MS_MethodDone
VAR_INPUT
END_VAR
bBusy := FALSE;
SUPER^.MS_MethodDone();
END_METHOD

METHOD PROTECTED MS_Ready
VAR_INPUT
END_VAR
eFcqFixtureStateInit := FIXTURE_INIT_CLAMP;
eFixtureState := UNIVERSAL_FIXTURE_IDLE;
END_METHOD

METHOD PROTECTED MS_Reset
VAR_INPUT
END_VAR
CASE eFcqFixtrueStateReset OF
	FIXTURE_RESET_CLAMP:
		fbClamp.MR_Reset();
		
		IF NOT fbClamp.Error THEN
			eFcqFixtrueStateReset := FIXTURE_RESET_COVER;
		END_IF
		
	FIXTURE_RESET_COVER:
		fbCover.MR_Reset();
		
		IF NOT fbCover.Error THEN
			eJigStateReset := FIXTURE_JIG_RESET_JIG_PUSHER;
			eFcqFixtrueStateReset := FIXTURE_RESET_DONE;
		END_IF
	
	FIXTURE_RESET_DONE:
		SUPER^.MS_Reset();
	
END_CASE
END_METHOD

METHOD PROTECTED MS_Uninitialized
VAR_INPUT
END_VAR
bNormLoaded := FALSE;

SUPER^.MS_Uninitialized();
END_METHOD

PROPERTY NormLoaded : REFERENCE TO BOOL
GET
NormLoaded REF= bNormLoaded;
END_GET
END_PROPERTY

PROPERTY NormLoadResults : REFERENCE TO E_FixtureLoadNormResult
GET
NormLoadResults REF= eNormLoadResult;
END_GET
END_PROPERTY

PROPERTY ref_Clamp : REFERENCE TO FB_FixtureClamp
GET
ref_Clamp REF= fbClamp;
END_GET
END_PROPERTY

PROPERTY ref_Cover : REFERENCE TO FB_DoubleCoilCylinder
GET
ref_Cover REF= fbCover;
END_GET
END_PROPERTY

PROPERTY StateExt : REFERENCE TO E_FixtureState
GET
StateExt REF= eFcqFixtureState;
END_GET
END_PROPERTY

METHOD PROTECTED StateMachine
VAR_INPUT
END_VAR
SUPER^.StateMachine();

CASE eFcqFixtureState OF
	E_FixtureState.FIXTURE_EXTENSION_COVER_ACTIVE:
		MS_CoverActive();
		
	E_FixtureState.FIXTURE_EXTENSION_COVER_ACTIVE_DONE:
		MS_CoverActiveDone();
		
	E_FixtureState.FIXTURE_EXTENSION_COVER_HOME:
		MS_CoverHome();
		
	E_FixtureState.FIXTURE_EXTENSION_COVER_HOME_DONE:
		MS_CoverHomeDone();
		
	E_FixtureState.FIXTURE_EXTENSION_CLAMP_HOLD:
		MS_ClampHold();
		
	E_FixtureState.FIXTURE_EXTENSION_CLAMP_HOLD_DONE:
		MS_ClampHoldDone();
		
	E_FixtureState.FIXTURE_EXTENSION_CLAMP_RELEASE:
		MS_ClampRelease();
		
	E_FixtureState.FIXTURE_EXTENSION_CLAMP_RELEASE_DONE:
		MS_ClampReleaseDone();
		
END_CASE
END_METHOD

END_FUNCTION_BLOCK

(* stored: Version 1.1.0.1, ProductVersion 3.1.4024.9
   POU FB_Fixture: Id {1f5616c3-fca8-44f4-90ea-3502d887ca35}, SpecialFunc None
   Folder Internal: Id {89905e4b-25ee-4002-a47a-6a9f53ba889b}
   Folder Properties: Id {9001b4ed-69b5-400d-a07a-e7f2c2b80c6d}
   Folder Parameters: Id {059479bb-d11f-4bc0-a5a4-37cc0bd06833}
   Folder References: Id {da1ea5a7-51fc-4fed-aa45-c2985cd1803c}
   Folder Status: Id {8925dcbe-dde5-4aab-a60e-bd9c6a8e07f6}
   Folder Requests: Id {5af6e07a-7e86-4f47-af0d-b4f8fd01c659}
   Folder StateMachine: Id {9bfbf726-05b0-4dd1-891c-b4123a6d3055}
   Folder StateMachineExt: Id {978d252b-71d8-4bad-ba39-11aafb528ed2}
   Property BatchEnd: Id {7ae70c46-2774-4c1a-8acf-fe19ae8336a7}
   Get Get: Id {52e0ac1a-33af-417f-babb-cae8ce13a424}
   Property ClampHold: Id {bb9cc494-dd3b-4bb8-85ba-5c9b93d58b47}
   Get Get: Id {1fe8fefa-a718-4f4e-9cbb-38a58c9c62ee}
   Property ClampSimulation: Id {8a133dc1-616a-4017-9769-70901fd91162}
   Get Get: Id {9cbe3a39-e212-4541-a61e-67701b3be4c3}
   Set Set: Id {eb200717-5617-4f22-ba76-ea55ffb20eda}
   Property CoverPositionActive: Id {7cbc9927-b5d6-4e8c-98e1-01dffcee8b7d}
   Get Get: Id {194a3eb5-ffde-40c2-850b-1651602fc1e0}
   Property CoverPositionHome: Id {57796bb9-397c-4633-8b98-f2e72ed82814}
   Get Get: Id {493eeb42-ad12-4b2b-86e0-f3b1de1d5ac6}
   Property CoverSimulation: Id {ab0f792a-7733-46a1-8654-0c7635b3c3df}
   Get Get: Id {2ca7d535-4767-42f1-af1e-4f07a9aff141}
   Set Set: Id {de660ab4-b58c-4986-986b-4c80a67b2af3}
   Property GoldenSampleMeasDone: Id {6c7216ca-79ca-4e69-bac6-0b839bf68b6f}
   Get Get: Id {01c662e9-3bad-4db8-af42-7ed5166c7fef}
   Property GoldenSampleMeasRequested: Id {d02965be-dbc9-4199-b8a4-0b40a0a508cc}
   Get Get: Id {a6f24009-de5e-494c-b07c-438ba489f35f}
   Property GoldenSampleResult: Id {155b26b2-b252-4565-bf9c-0ee8a2511d7d}
   Get Get: Id {3e276241-7ad1-464d-88e1-6ce337757dd5}
   Property GSampleId: Id {5a4e4fb4-5ef3-46f7-a2af-32f5592c659b}
   Get Get: Id {edf7a59e-a792-4c06-8e67-593855f22936}
   Method M_MeasurementClient: Id {059ce93c-3f97-4c14-8662-ce1aed6607e3}
   Property MeasurementResultExt: Id {1bdec847-179d-43eb-8460-536d6a3998d5}
   Get Get: Id {b69dadf1-39ba-451a-a16a-df5cdab8288c}
   Method MR_ClampHold: Id {a84ca68a-16b4-400c-9ce2-7d99e61055be}
   Method MR_ClampRelease: Id {dfd2a2c8-ea94-458c-ae2e-64fdd3d66f48}
   Method MR_CoverActive: Id {6d774f73-8e6e-4ce2-a32a-00b2ea22d282}
   Method MR_CoverActiveAndJigOpen: Id {1319735a-57dc-45b7-becf-ba6497c01954}
   Method MR_CoverHome: Id {dfa8dcbb-576d-487e-8a6f-0c53ee3e58ce}
   Method MR_CoverHomeAndJigClose: Id {e9860585-0df9-4174-a642-ea6c27a06bb0}
   Method MR_GSampleMeas: Id {980716de-93a1-4338-9c33-85c48e4f962b}
   Method MR_LoadNorm: Id {79191bd3-f77a-4cdf-8045-0dc7ee99e711}
   Method MR_Reset: Id {c571d1bc-8f20-43e9-a102-a8f141fdbeda}
   Method MS_Aborting: Id {387b38da-395d-4e10-a40e-06c55fcdec85}
   Method MS_ClampHold: Id {6ebdcd0b-68e1-413a-9e37-7f1fb0be3561}
   Method MS_ClampHoldDone: Id {8f7929c3-1e42-4012-af91-c364c00acd5a}
   Method MS_ClampRelease: Id {3d13e849-33a7-4d47-a5f2-1f759792fe36}
   Method MS_ClampReleaseDone: Id {63a4cdff-c2b0-4cf8-a872-93ada06e4273}
   Method MS_CoverActive: Id {a56ced19-3082-4311-abac-e92652f9ed9a}
   Method MS_CoverActiveAndJigOpen: Id {90abf1f6-ca5e-49d7-8b90-09f89011bbaf}
   Method MS_CoverActiveAndJigOpenDone: Id {d093094d-8171-432d-a4a6-d3504c27699e}
   Method MS_CoverActiveDone: Id {f8def135-901d-4216-9011-e046695a85bf}
   Method MS_CoverHome: Id {0c8fafe9-0ded-453a-bf78-970d64e717e0}
   Method MS_CoverHomeAndJigClose: Id {20d3a174-d73c-421a-a3b9-6b6fd09fe426}
   Method MS_CoverHomeAndJigCloseDone: Id {599a3eed-a5cd-4d13-a6bd-7c9d89f9bfcf}
   Method MS_CoverHomeDone: Id {b521ecfd-d9ad-4f39-8c4c-aacc00c34c9d}
   Method MS_Extension: Id {1cca78b6-1bb8-4c47-a47a-fea2b5aee859}
   Method MS_GSampleMeas: Id {c1fd972d-0566-46b7-b157-7b3d8fc28123}
   Method MS_GSampleMeasDone: Id {d32c2fb1-14c5-413b-aa70-f01436f5fd48}
   Method MS_Initializing: Id {9307c2c4-2f46-48f3-a2d6-5139d9bd71d4}
   Method MS_LoadNorm: Id {7c00fcea-1aaa-40c0-ad3f-0a8234d51dac}
   Method MS_LoadNormDone: Id {d278ec86-3588-4b3e-bdb6-3e68ec6597d1}
   Method MS_MethodDone: Id {42d7f3dd-9b70-45ca-abe5-ec05fed60233}
   Method MS_Ready: Id {1a89915f-d569-41db-8855-9aef83440988}
   Method MS_Reset: Id {70f992d0-ec66-43cd-bef0-00b72e8b0896}
   Method MS_Uninitialized: Id {e5476f48-7990-48bb-ada3-68d5c93cc0a7}
   Property NormLoaded: Id {66e6b5d7-1834-499b-8eaa-8a84a381c494}
   Get Get: Id {641b316e-c574-4db6-9b16-93449624139e}
   Property NormLoadResults: Id {96673ae4-51ed-40f1-a0f8-282fa6205524}
   Get Get: Id {2afe6081-f443-4ee5-a3f5-bebebf67c8a3}
   Property ref_Clamp: Id {49c505e2-f58a-4747-a541-916ae5c865ce}
   Get Get: Id {7492b162-d196-4e81-8563-389f913f9e06}
   Property ref_Cover: Id {3a7ae8d7-9bf1-4722-a1ab-863056ed0be3}
   Get Get: Id {bfa92e06-b06b-4e1d-a788-ee3e4e34ba93}
   Property StateExt: Id {d0b38adb-6abf-4c49-89de-54a4ce30dc41}
   Get Get: Id {0cc28eb4-16ca-4d10-8f82-953680a7397b}
   Method StateMachine: Id {f2d90476-4ae2-45da-a431-68f71ef3d71d} *)
